(* CoDeSys 2.3.9.47 project: Test.pro *)
(* Libraries: Standard.lib 20.5.14 08:13:26, Iecsfc.lib 30.1.13 13:05:12, SYSLIBCALLBACK.LIB 30.1.13 13:05:12 *)

(* PLC configuration (modules and I/O channels)
K-Bus [K_Bus] node 0, in %IB0 out %QB0 {KbusBusMode = 1; KbusCycleTime = 10000; KbusThreadPriority = 0; KbusSetOutputsToZeroOnApplicationStop = 1}
Modbus variables [PFC200MODBUS] node 1, in %IB0 out %QB0 {PlcStopBehaviour = 1; FiledbusErrorBehaviour = 1; TcpOperation = 1; TcpPort = 502; TcpTimeout = 600; UdpOperation = 1; UdpPort = 502; RtuOperation = 0; NodeId = 1; ResponseTimeout = 5000; Interface = 0; Baud = 115200; StopBits = 1; Parity = 1; FlowCtrl = 0; PhysInterface = 0}
Modbus-Master [MB_MASTER] node 2, in %IB0 out %QB0
*)

(* Task configuration *)
TASK NewTask (PRIORITY := 31, INTERVAL := T#1000ms);
	Test();
END_TASK

(* POU SWITCHING RELAIS/Test, ST *)
PROGRAM Test
VAR

	Test :fbSwitchRelaysOnOffGrid;
	a: REAL;
END_VAR
Test(
	r_Off_Grid_Bus_Frequency:= a ,
	r_Off_Grid_Bus_Voltage:= 250,
	r_On_Grid_Start_Frequency:= 51,
	r_On_Grid_Start_Delay_Time:= 2000,
	r_On_Grid_Minimal_On_Time:= 2000 ,
	r_Off_Grid_Start_Frequency:= 49,
	r_Off_Grid_Start_Delay_Time:= 2000,
	r_Switch_Gap_Time:= 2000,
	r_Off_Grid_Minimal_On_Time:= 2000);
END_PROGRAM

(* POU SWITCHING RELAIS/fbSwitchRelaysOnOffGrid, SFC *)
FUNCTION_BLOCK fbSwitchRelaysOnOffGrid
VAR_INPUT

	r_Off_Grid_Bus_Frequency						:	REAL;
	r_Off_Grid_Bus_Voltage							:	REAL;
	r_On_Grid_Start_Frequency						:	REAL;
	r_On_Grid_Start_Delay_Time					:	REAL;
	r_On_Grid_Minimal_On_Time					:	REAL;
	r_Off_Grid_Start_Frequency						:	REAL;
	r_Off_Grid_Start_Delay_Time					:	REAL;
	r_Switch_Gap_Time								: 	REAL;		(* Time between on and off grid relay switching (dead bus gap) *)
	r_Off_Grid_Minimal_On_Time					:	REAL;

END_VAR
VAR_OUTPUT

	r_On_Grid_Relay									:	BOOL;
	r_Off_Grid_Relay									:	BOOL;

END_VAR
VAR

	r_Checked_On_Grid_Start_Frequency			:	REAL;
	r_Checked_Off_Grid_Start_Frequency			:	REAL;

	t_On_Grid_Start_Delay_Timer					:	TON;
	t_Off_Grid_Start_Delay_Timer					:	TON;


END_VAR
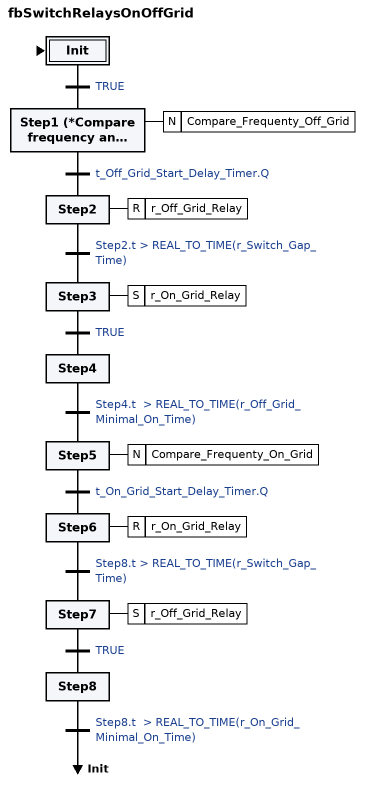
INITIAL_STEP Init:
END_STEP
TRANSITION FROM Init TO Step1 (*Compare frequency and voltage *) := TRUE;
END_TRANSITION
STEP Step1 (*Compare frequency and voltage *):
	Compare_Frequenty_Off_Grid(N);
END_STEP
TRANSITION FROM Step1 (*Compare frequency and voltage *) TO Step2 := t_Off_Grid_Start_Delay_Timer.Q;
END_TRANSITION
STEP Step2:
	r_Off_Grid_Relay(R);
END_STEP
TRANSITION FROM Step2 TO Step3 := Step2.t > REAL_TO_TIME(r_Switch_Gap_Time);
END_TRANSITION
STEP Step3:
	r_On_Grid_Relay(S);
END_STEP
TRANSITION FROM Step3 TO Step4 := TRUE;
END_TRANSITION
STEP Step4:
END_STEP
TRANSITION FROM Step4 TO Step5 := Step4.t  > REAL_TO_TIME(r_Off_Grid_Minimal_On_Time);
END_TRANSITION
STEP Step5:
	Compare_Frequenty_On_Grid(N);
END_STEP
TRANSITION FROM Step5 TO Step6 := t_On_Grid_Start_Delay_Timer.Q;
END_TRANSITION
STEP Step6:
	r_On_Grid_Relay(R);
END_STEP
TRANSITION FROM Step6 TO Step7 := Step8.t > REAL_TO_TIME(r_Switch_Gap_Time);
END_TRANSITION
STEP Step7:
	r_Off_Grid_Relay(S);
END_STEP
TRANSITION FROM Step7 TO Step8 := TRUE;
END_TRANSITION
STEP Step8:
END_STEP
TRANSITION FROM Step8 TO Init := Step8.t  > REAL_TO_TIME(r_On_Grid_Minimal_On_Time);
END_TRANSITION
END_FUNCTION_BLOCK
ACTION Compare_Frequencies:
(* Off grid frequency should by higher than on grid frequency to prevent pendel behaviour of states *)

IF r_Off_Grid_Start_Frequency > r_On_Grid_Start_Frequency THEN

	r_Checked_Off_Grid_Start_Frequency := r_Off_Grid_Start_Frequency;
	r_Checked_On_Grid_Start_Frequency := r_On_Grid_Start_Frequency;

ELSE

	r_Checked_Off_Grid_Start_Frequency := r_Off_Grid_Start_Frequency;
	r_Checked_On_Grid_Start_Frequency := r_Off_Grid_Start_Frequency;

END_IF
END_ACTION
ACTION Compare_Frequenty_Off_Grid:
t_Off_Grid_Start_Delay_Timer(
	IN:= r_Off_Grid_Bus_Frequency > r_Checked_Off_Grid_Start_Frequency AND r_Off_Grid_Bus_Voltage > 150,
	PT:= REAL_TO_TIME(r_On_Grid_Start_Delay_Time));
END_ACTION
ACTION Compare_Frequenty_On_Grid:
t_On_Grid_Start_Delay_Timer(
	IN:= r_Off_Grid_Bus_Frequency < r_Checked_On_Grid_Start_Frequency,
	PT:= REAL_TO_TIME(r_Off_Grid_Start_Delay_Time));
END_ACTION
